PROGRAM MAIN
VAR
   MuteLCfromHMI AT %I* : BOOL;
END_VAR

END_PROGRAM

(* stored: Version 1.1.0.1, ProductVersion 3.1.4024.5
   POU MAIN: Id {98ae381b-1fae-4503-a3b8-1900850a68a0}, SpecialFunc None *)
